FUNCTION_BLOCK WithOutputs (* Only UPDATE updates the data inputs *)
  (* Standard: 61499-2 *)
  (* Version 1.0, 2023-03-07, AK115394 *)
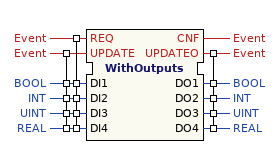
  EVENT_INPUT
    REQ WITH DI1, DI2, DI3, DI4;
    UPDATE WITH DI1, DI2, DI3, DI4;
  END_EVENT
  EVENT_OUTPUT
    CNF;
    UPDATEO WITH DO1, DO3, DO2, DO4;
  END_EVENT
  VAR_INPUT
    DI1 : BOOL;
    DI2 : INT;
    DI3 : UINT;
    DI4 : REAL;
  END_VAR
  VAR_OUTPUT
    DO1 : BOOL := 1;
    DO2 : INT := -42;
    DO3 : UINT := 21;
    DO4 : REAL := 3.14;
  END_VAR
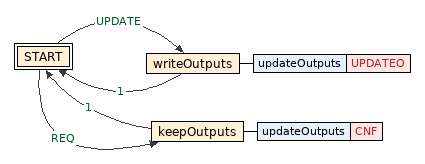
  EC_STATES
    START; (* Initial State *)
    writeOutputs : updateOutputs -> UPDATEO;
    keepOutputs : updateOutputs -> CNF;
  END_STATES
  EC_TRANSITIONS
    writeOutputs TO START := 1;
    START TO writeOutputs := UPDATE;
    START TO keepOutputs := REQ;
    keepOutputs TO START := 1;
  END_TRANSITIONS
  ALGORITHM updateOutputs IN ST:
DO1 := DI1;
DO2 := DI2;
DO3 := DI3;
DO4 := DI4;
  END_ALGORITHM
END_FUNCTION_BLOCK
